TYPE IRecipe :
STRUCT
	bCreate:BOOL;
	bSave:BOOL;
	bLoad:BOOL;

     
END_STRUCT
END_TYPE

(* stored: Version 1.1.0.1, ProductVersion 3.1.4024.9
   DUT IRecipe: Id {f3d25308-9369-4ecd-8e75-48dae62282c3} *)
